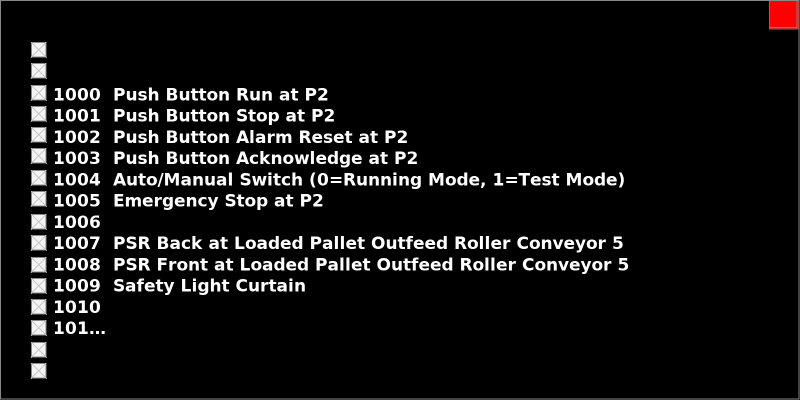
VISUALIZATION P2_DI1  // 800x400, background image 
    ImageSwitcher (31,42 15x15), variable: InputOutput_GVL.Digital_Input[1], behaviour: TOGGLE
    Label (50,16 724x391), "1000 Push Button Run at P2 1001 Push Button Stop at P2 1002 Push Button Alarm Reset at P2 1003 Push Button Acknowledge at P2 1004 Auto/Manual Switch (0=Running Mode, 1=Test Mode) 1005 Emergency Stop at P2 1006 1007 PSR Back at Loaded Pallet Outfeed Roller Conveyor 5 1008 PSR Front at Loaded Pallet Outfeed Roller Conveyor 5 1009 Safety Light Curtain 1010 1011 1012 1013 PSR Back at Detect Loaded Pallet Buffer Roller Conv 2 1014 PSR Front at Detect Loaded Pallet Buffer Roller Conv 2 1015 Feedback Loaded Pallet Outfeed Roller Conveyor 5 is Running"
    ImageSwitcher (31,63 15x15), variable: InputOutput_GVL.Digital_Input[2], behaviour: TOGGLE
    ImageSwitcher (31,85 15x15), variable: InputOutput_GVL.Digital_Input[3], behaviour: TOGGLE
    ImageSwitcher (31,106 15x15), variable: InputOutput_GVL.Digital_Input[4], behaviour: TOGGLE
    ImageSwitcher (31,127 15x15), variable: InputOutput_GVL.Digital_Input[5], behaviour: TOGGLE
    ImageSwitcher (31,148 15x15), variable: InputOutput_GVL.Digital_Input[6], behaviour: TOGGLE
    ImageSwitcher (31,170 15x15), variable: InputOutput_GVL.Digital_Input[7], behaviour: TOGGLE
    ImageSwitcher (31,191 15x15), variable: InputOutput_GVL.Digital_Input[8], behaviour: TOGGLE
    ImageSwitcher (31,214 15x15), variable: InputOutput_GVL.Digital_Input[9], behaviour: TOGGLE
    ImageSwitcher (31,235 15x15), variable: InputOutput_GVL.Digital_Input[10], behaviour: TOGGLE
    ImageSwitcher (31,257 15x15), variable: InputOutput_GVL.Digital_Input[11], behaviour: TOGGLE
    ImageSwitcher (31,278 15x15), variable: InputOutput_GVL.Digital_Input[12], behaviour: TOGGLE
    ImageSwitcher (31,299 15x15), variable: InputOutput_GVL.Digital_Input[13], behaviour: TOGGLE
    ImageSwitcher (31,320 15x15), variable: InputOutput_GVL.Digital_Input[14], behaviour: TOGGLE
    ImageSwitcher (31,342 15x15), variable: InputOutput_GVL.Digital_Input[15], behaviour: TOGGLE
    ImageSwitcher (31,363 15x15), variable: InputOutput_GVL.Digital_Input[16], behaviour: TOGGLE
    Button (769,-1 30x30), image: VisuSymbols.Symbols.Wrong
        OnMouseClick: CloseDialog Dialog=P2_DI1, Result=OK, NumpadKeypadSet=True
END_VISUALIZATION

(* stored: Version 1.1.0.1, ProductVersion 3.1.4024.12
   Visu P2_DI1: Id {204e4367-3b02-4dfe-b0ec-0f6e5f4f0c20} *)
